//-----------------------------------------------------------------------------------------
//
//                  				ST_Log
//
//								Structure Log 			
//-----------------------------------------------------------------------------------------
//
//Auteur: G.GOETZ (inspired by S.MANTZER)
//Création: 04.02.2026
//Dernière modification : 04.02.2026 (G.GOETZ)
//       			
//-----------------------------------------------------------------------------------------
//
//     							Liste des modifications  	
//
// 04.02.2026 (G.GOETZ) -> Création		
//-----------------------------------------------------------------------------------------

TYPE ST_Log :
STRUCT
	
	(** STRING **)
	strLogDateTime : STRING[50] ; // Date and Time to Log
	strLogTxt : STRING[255] ; // Text to Log
	
END_STRUCT
END_TYPE

(* stored: Version 1.1.0.1, ProductVersion 3.1.4024.13
   DUT ST_Log: Id {2ae9a3c1-ee3a-42cb-b1eb-1c2c76ea3634} *)
